// TwinCAT 3 PLC project SAmpleVisionRefactoringSimple
// ProgramVersion: 3.1.4024.0
// libraries:
//   Tc2_Standard, * (Beckhoff Automation GmbH)
//   Tc2_System, * (Beckhoff Automation GmbH)
//   Tc3_Module, * (Beckhoff Automation GmbH)
// project tree:
//   DUTs/ LED1904.TcDUT
//   DUTs/Vision/ ST_CenterPosition.TcDUT, ST_ColorSimularity.TcDUT, ST_Conture.TcDUT, ST_PositionBounds.TcDUT, ST_PositionDeviation.TcDUT, ST_PositionXY.TcDUT, ST_ThresholdData.TcDUT
//   GVLs/ Globale_Definitionen.TcGVL, Globale_Kamera_Variablen.TcGVL
//   / PlcTask.TcTTO
//   POUs/ Camera.TcPOU, MAIN.TcPOU
// (motion and I/O tree: see PLC project plc1)
// real-time tasks:
//   TASK PlcTask: cycle T#10ms, priority 20, ADS port 350
//   TASK PlcTask1: cycle T#10ms, priority 21, ADS port 351
//   TASK PlcTask2: cycle T#10ms, priority 22, ADS port 352

CONFIGURATION SAmpleVisionRefactoringSimple
    RESOURCE PLC ON TwinCAT3
        TASK PlcTask(INTERVAL := T#10ms, PRIORITY := 22);
        PROGRAM MAIN WITH PlcTask : MAIN;
    END_RESOURCE
END_CONFIGURATION

// ---- DUTs/LED1904.TcDUT
TYPE LED1904 :
STRUCT
	bInput1:BOOL;
	bInput2:BOOL;
	bInput3:BOOL;
	bInput4:BOOL;
	bDiag1:BOOL;
	bDiag2:BOOL;
	bDiag3:BOOL;
	bDiag4:BOOL;
END_STRUCT
END_TYPE

// ---- DUTs/Vision/ST_CenterPosition.TcDUT
TYPE ST_CenterPosition :
STRUCT
  Input : ST_PositionXY;
  Diagnose : ST_PositionXY;
END_STRUCT
END_TYPE

// ---- DUTs/Vision/ST_ColorSimularity.TcDUT
TYPE ST_ColorSimularity :
STRUCT
	aRefColor :	TcVnPoint3_LREAL;
	aRefColorGreen : TcVnPoint3_LREAL	:= [130, 230, 0];
	aRefColorRed : TcVnPoint3_LREAL	:= [255, 255, 255];
	aRefColorPrismError :	TcVnPoint3_LREAL := [135, 150, 105];
	fVariance :	REAL := 0.10;
	fLuminanceWeight :	REAL := 0.1;
END_STRUCT
END_TYPE

// ---- DUTs/Vision/ST_Conture.TcDUT
TYPE ST_Conture :
STRUCT
	fAreaMin : REAL;		(*Mindestfläche der zufindenden LED*)
	fAreaMax : REAL;		(*Mindestfläche der zufindenden LED*)
	fHeightMin : REAL;		(*Mindesthöhe der zufindenden LED*)
	fHeightMax : REAL;		(*Maximalhöhe der zufindenden LED*)
	fWidthMax : REAL;		(*Maximalhöhe der zufindenden LED*)
END_STRUCT
END_TYPE

// ---- DUTs/Vision/ST_PositionBounds.TcDUT
TYPE ST_PositionBounds :
STRUCT
  stDeviation : ST_PositionDeviation; 
	aCenterReferenceCoordinatesXY	: ARRAY  [1..8] OF TcVnPoint2_REAL;
  aCenterPosition : ARRAY[1..4] OF ST_CenterPosition;  
END_STRUCT
END_TYPE

// ---- DUTs/Vision/ST_PositionDeviation.TcDUT
TYPE ST_PositionDeviation :
STRUCT
  nLower : UINT;
	nUpper : UINT;
END_STRUCT
END_TYPE

// ---- DUTs/Vision/ST_PositionXY.TcDUT
TYPE ST_PositionXY :
STRUCT
  X : REAL;
  Y : REAL;
END_STRUCT
END_TYPE

// ---- DUTs/Vision/ST_ThresholdData.TcDUT
TYPE ST_ThresholdData :
STRUCT
	fThreshold : LREAL;	(* fixed threshold (unused if dynamic thresholding is selected) *)
	fMaxValue :	LREAL;	(* maximum pixel value *)
END_STRUCT
END_TYPE

// ---- GVLs/Globale_Definitionen.TcGVL
{attribute 'Tc2GvlVarNames'}
VAR_GLOBAL
	FileName: STRING := 'C:\TwinSAFE\TestErgebnisse\EL1904\TestLog_EL1904_';
	StartUp_Wait_Time: TIME := t#3s;
	ShutDown_Wait_Time : TIME := T#1S;
	Kamera_Wait_Time: TIME := T#2S;
	Prisma_Wait_Time:  TIME := T#3S;
	Seriell_Wait_Time: TIME := T#1S;
	KameraBeleuchtungFaktorWarteZeit:UINT:=8;
	Kopfzeile: STRING(255);
	TesterArray: ARRAY[0..7] OF STRING ;
	EtherCATAmsNetID: T_AmsNetId := '172.16.3.218.2.1';
	EL1904port: T_AmsPort := 1024;
	EL6900port: T_AmsPort := 1010;
	OutputWait_Time: TIME := t#5s;
	Color_Rot : DWORD := 16#000000FF;
	Color_Gruen : DWORD := 16#00007F00;
	Color_Weiss : DWORD := 16#00FFFFFF;
	Color_Visu : DWORD := 16#00FFFFFF;
	VoltagePowerContacts20Vunder : UINT := 21300; (* 0V = 0, 30V = 32767  1092 pro Volt  20V = 21845*)
	VoltagePowerContacts20Vover : UINT := 22300; (* 0V = 0, 30V = 32767  1092 pro Volt  20V = 21845*)
	VoltagePowerContacts24Vunder : UINT := 25900; (* 0V = 0, 30V = 32767  1092 pro Volt  24V = 26213*)
	VoltagePowerContacts24Vover : UINT := 26700; (* 0V = 0, 30V = 32767  1092 pro Volt  24V = 26213*)
	VoltagePowerContacts30Vunder : UINT := 32200; (* 0V = 0, 30V = 32767  1092 pro Volt  30V = 32767*)
	VoltagePowerContacts30Vover : UINT := 32767; (* 0V = 0, 30V = 32767  1092 pro Volt  30V = 32767*)
	LogFileSerialNumber: UDINT;
	Artikel : UDINT := 70931;
//	SafetyProg1: T_MaxString := 'C:\TwinSAFE\Programm\EL\Automated_EL1904\1_SafetyProgramCRC';
//	SafetyCRC1: WORD := 17617;
	SafetyProg65534: T_MaxString := 'C:\TwinSAFE\Programm\EL\Automated_EL1904\65534_SafetyProgramCRC';
	SafetyCRC65534: WORD := 65346;
END_VAR

// ---- GVLs/Globale_Kamera_Variablen.TcGVL
{attribute 'qualified_only'}
VAR_GLOBAL
	//TestVariablen
	bStopStepPrismaDetection:BOOL:=FALSE;
	bStopStepAllLedOn:BOOL:=FALSE;
	bEinrichtBetrieb:BOOL:=FALSE;
	bNextStepEinrichtbetrieb:BOOL:=FALSE;
	bPrismaOk:BOOL:=FALSE;
	bPrismaNotOK:BOOL:=FALSE;
	
	//Kamera aktiv
	bKameraAktiv:BOOL:=TRUE;
	
	//erkannte LEDs
	bLED_TermXOn		: ARRAY  [1..8] OF LED1904;
	iDetectedLED			: INT:=0;
	iStartDetectedLED		: INT:=1;
	
	// Color Simularity
//	aRefColor					:	TcVnPoint3_LREAL;
//	aRefColorGreen				:	TcVnPoint3_LREAL	:= [130, 230, 0];
//	aRefColorRed				:	TcVnPoint3_LREAL	:= [255, 255, 255];
//	aRefColorPrismError			:	TcVnPoint3_LREAL	:= [135, 150, 105];
//	fVariance					:	REAL := 0.10;
//	fLuminanceWeight			:	REAL := 0.1;
  stColorSimularity : ST_ColorSimularity;
  
  
	
	//Threshold
  stThreshold : ST_ThresholdData; 
  stThresholdGreenLed : ST_ThresholdData := (fThreshold := 10, fMaxValue := 255); 
  stThresholdRedLed : ST_ThresholdData := (fThreshold := 15, fMaxValue := 255); 
  stThresholdPrism : ST_ThresholdData := (fThreshold := 185, fMaxValue := 255); 
	
	//Konturen zeichnen
  stConture : ST_Conture := (fAreaMin := 1200,fAreaMax := 3000, fHeightMin := 30, fHeightMax := 70, fWidthMax:= 70 );
  stContureLED : ST_Conture := (fAreaMin := 1200,fAreaMax := 3000, fHeightMin := 30, fHeightMax := 70, fWidthMax:= 90 );
  stConturePrisma : ST_Conture := (fAreaMin := 450,fAreaMax := 900, fHeightMin := 20, fHeightMax := 70, fWidthMax:= 70 );
	
	// Positionsgrenzen
//	uiLowerPosDeviation:UINT:=10;
//	uiUpperPosDeviation:UINT:=10;
//	aCenterReferenceCoordinatesXY	: ARRAY  [1..8] OF TcVnPoint2_REAL;
//	CenterXPosInput1:REAL:=46;
//	CenterYPosInput1:REAL:=36;
//	CenterXPosInput2:REAL:=119;
//	CenterYPosInput2:REAL:=33;
//	CenterXPosInput3:REAL:=46;
//	CenterYPosInput3:REAL:=87;
//	CenterXPosInput4:REAL:=120;
//	CenterYPosInput4:REAL:=87;
//	CenterXPosDiag1:REAL:=46;
//	CenterYPosDiag1:REAL:=139;
//	CenterXPosDiag2:REAL:=114;
//	CenterYPosDiag2:REAL:=137;
//	CenterXPosDiag3:REAL:=45;
//	CenterYPosDiag3:REAL:=192;
//	CenterXPosDiag4:REAL:=124;
//	CenterYPosDiag4:REAL:=192;
  
  stPositionBounds : ST_PositionBounds;


//PositionBounds.aCenterPosition[1].Diagnose.X
  
  
	// Region of Interrest
	nXposPrisma			:	UDINT:=1514;
	nYposPrisma			:	UDINT:=892;
	nROIWidth			:	UDINT:=170;
	nROIHeight			:	UDINT:=220;
	
	// Beleuchtung EL2595
	bLedOn AT%Q* :BOOL;
	uiOutputCurrent AT%Q*:UINT;
	bLedReset AT%Q*:BOOL;
	bLedWarning AT%I*:BOOL;
	bLedError AT%I*:BOOL;	
	uiOutputCurrentEinrichtbertieb:UINT:=300;
END_VAR

// ---- POUs/MAIN.TcPOU
PROGRAM MAIN
VAR
END_VAR

END_PROGRAM

// ---- POUs/Camera.TcPOU
PROGRAM Camera
VAR
	
  hr : HRESULT;
  fbCameraControl :	FB_VN_GevCameraControl; //SymbolInitialization  verlinken!
	eState : ETcVnCameraState;
	
	ipImgIn :	ITcVnImage;
	ipImgRoi :   ITcVnImage;
	ipImgRotated :   ITcVnImage;
	ipImgConvertColorSpace : 	ITcVnImage;
	ipImgColorSimilarity :	ITcVnImage;
	ipImgThreshold :	ITcVnImage;
	ipImgResult :	ITcVnImage;
	
	ipImg_Eingangsbild : ITcVnDisplayableImage;
	ipImg_Ausgeschnitten : ITcVnDisplayableImage;
	ipImg_Gedreht :	ITcVnDisplayableImage;
	ipImg_Farbbild : ITcVnDisplayableImage;
	ipImg_Farbauswahl :	ITcVnDisplayableImage;
	ipImg_Schwellwert_Farbauswahl :	ITcVnDisplayableImage;
	ipImg_Ergebnis :	ITcVnDisplayableImage;
	
	
	// Region of Interrest
	nXposTerm1 : UDINT;
	nYposTerm1 : UDINT;
	nROIWidth :	UDINT;
	nROIHeight : UDINT;
	
	// Get Center 
	aCenterCoordinatesXY : ARRAY[1..8] OF TcVnPoint2_REAL;
	
	aWhite : TcVnVector4_LREAL :=	[255,255,255];
	aBlack : TcVnVector4_LREAL :=	[0,0,0];
	aRed : TcVnVector4_LREAL := 	[255,0,0];
	aGreen : TcVnVector4_LREAL :=	[0,255,0];
	aBlue :	TcVnVector4_LREAL :=	[0,0,255];
	aOrange :	TcVnVector4_LREAL :=	[255,150,0];
END_VAR

VAR
  // Init
  bInitPositionBoundsDone : BOOL := FALSE;
  nClearByteLength : UDINT;
END_VAR

// Init
InitPositionBounds(bInitPositionBoundsDone, Globale_Kamera_Variablen.stPositionBounds);


// Position zum Zuschneiden des Prismas aus der Visu übergeben
nXposTerm1 := Globale_Kamera_Variablen.nXposPrisma;
nYposTerm1 := Globale_Kamera_Variablen.nYposPrisma;
nROIWidth := Globale_Kamera_Variablen.nROIWidth;
nROIHeight := Globale_Kamera_Variablen.nROIHeight;

// Kamera Kontroll Status Maschine
eState := fbCameraControl.GetState();
//eState := fbFileSource.GetState();

CASE eState OF
	
  TCVN_CS_INITIAL, TCVN_CS_OPENING, TCVN_CS_OPENED, TCVN_CS_STARTACQUISITION:
    hr := fbCameraControl.StartAcquisition();
	
  TCVN_CS_ACQUIRING:
    hr := fbCameraControl.GetCurrentImage(ipImgIn);
	
    IF SUCCEEDED(hr) AND ipImgIn <> 0 THEN
      VisionLedDetecting(); 		(*Methoden Aufruf*)
    
      hr := F_VN_TransformIntoDisplayableImage(ipImgIn, ipImg_Eingangsbild, S_OK);
      hr := F_VN_TransformIntoDisplayableImage(ipImgRoi, ipImg_Ausgeschnitten, S_OK);
      hr := F_VN_TransformIntoDisplayableImage(ipImgRotated, ipImg_Gedreht, S_OK);
      hr := F_VN_TransformIntoDisplayableImage(ipImgConvertColorSpace, ipImg_Farbbild, S_OK);
      hr := F_VN_TransformIntoDisplayableImage(ipImgColorSimilarity, ipImg_Farbauswahl, S_OK);
      hr := F_VN_TransformIntoDisplayableImage(ipImgThreshold, ipImg_Schwellwert_Farbauswahl, S_OK);
      hr := F_VN_TransformIntoDisplayableImage(ipImgResult, ipImg_Ergebnis, S_OK);
      
    END_IF

  // Freigeben der Bilder sonst kann es zum Page Fault kommen
    Tc3_Module.FW_SafeRelease(ADR(ipImgIn));
    Tc3_Module.FW_SafeRelease(ADR(ipImgRoi));
    Tc3_Module.FW_SafeRelease(ADR(ipImgRotated));
    Tc3_Module.FW_SafeRelease(ADR(ipImgConvertColorSpace));
    Tc3_Module.FW_SafeRelease(ADR(ipImgColorSimilarity));
    Tc3_Module.FW_SafeRelease(ADR(ipImgThreshold));
    Tc3_Module.FW_SafeRelease(ADR(ipImgResult));

  TCVN_CS_ERROR:
    //hr := fbFileSource.Reset();
    hr := fbCameraControl.Reset();
    
  END_CASE

//Positionen der Mittelpunktskoordinaten aus der Visu übernehmen
GetCenterPositionFromVisu(Globale_Kamera_Variablen.stPositionBounds);
	
//Detectiere LEDs	
//Diag1 LED
Globale_Kamera_Variablen.iStartDetectedLED:=1;
DetectLedCoordinate(
    nStartDetectedLED:= Globale_Kamera_Variablen.iStartDetectedLED, 
    nDetectedLED:= Globale_Kamera_Variablen.iDetectedLED, 
    nLedNumber:= 5, 
    aCenterCoordinatesXY:= aCenterCoordinatesXY[Globale_Kamera_Variablen.iStartDetectedLED], 
    stPositionBounds:= Globale_Kamera_Variablen.stPositionBounds, 
    Detected:= Globale_Kamera_Variablen.bLED_TermXOn[1].bDiag1);

//Diag2 LED
Globale_Kamera_Variablen.iStartDetectedLED:=1;
DetectLedCoordinate(
    nStartDetectedLED:= Globale_Kamera_Variablen.iStartDetectedLED, 
    nDetectedLED:= Globale_Kamera_Variablen.iDetectedLED, 
    nLedNumber:= 6, 
    aCenterCoordinatesXY:= aCenterCoordinatesXY[Globale_Kamera_Variablen.iStartDetectedLED], 
    stPositionBounds:= Globale_Kamera_Variablen.stPositionBounds, 
    Detected:= Globale_Kamera_Variablen.bLED_TermXOn[1].bDiag2);

//Diag3 LED
Globale_Kamera_Variablen.iStartDetectedLED:=1;
DetectLedCoordinate(
    nStartDetectedLED:= Globale_Kamera_Variablen.iStartDetectedLED, 
    nDetectedLED:= Globale_Kamera_Variablen.iDetectedLED, 
    nLedNumber:= 7, 
    aCenterCoordinatesXY:= aCenterCoordinatesXY[Globale_Kamera_Variablen.iStartDetectedLED], 
    stPositionBounds:= Globale_Kamera_Variablen.stPositionBounds, 
    Detected:= Globale_Kamera_Variablen.bLED_TermXOn[1].bDiag3);


//Diag4 LED
Globale_Kamera_Variablen.iStartDetectedLED:=1;
DetectLedCoordinate(
    nStartDetectedLED:= Globale_Kamera_Variablen.iStartDetectedLED, 
    nDetectedLED:= Globale_Kamera_Variablen.iDetectedLED, 
    nLedNumber:= 8, 
    aCenterCoordinatesXY:= aCenterCoordinatesXY[Globale_Kamera_Variablen.iStartDetectedLED], 
    stPositionBounds:= Globale_Kamera_Variablen.stPositionBounds, 
    Detected:= Globale_Kamera_Variablen.bLED_TermXOn[1].bDiag4);

//Input1 LED
Globale_Kamera_Variablen.iStartDetectedLED:=1;
DetectLedCoordinate(
    nStartDetectedLED:= Globale_Kamera_Variablen.iStartDetectedLED, 
    nDetectedLED:= Globale_Kamera_Variablen.iDetectedLED, 
    nLedNumber:= 1, 
    aCenterCoordinatesXY:= aCenterCoordinatesXY[Globale_Kamera_Variablen.iStartDetectedLED], 
    stPositionBounds:= Globale_Kamera_Variablen.stPositionBounds, 
    Detected:= Globale_Kamera_Variablen.bLED_TermXOn[1].bInput1);

//Input2 LED
Globale_Kamera_Variablen.iStartDetectedLED:=1;
DetectLedCoordinate(
    nStartDetectedLED:= Globale_Kamera_Variablen.iStartDetectedLED, 
    nDetectedLED:= Globale_Kamera_Variablen.iDetectedLED, 
    nLedNumber:= 2, 
    aCenterCoordinatesXY:= aCenterCoordinatesXY[Globale_Kamera_Variablen.iStartDetectedLED], 
    stPositionBounds:= Globale_Kamera_Variablen.stPositionBounds, 
    Detected:= Globale_Kamera_Variablen.bLED_TermXOn[1].bInput2);

//Input3 LED
Globale_Kamera_Variablen.iStartDetectedLED:=1;
DetectLedCoordinate(
    nStartDetectedLED:= Globale_Kamera_Variablen.iStartDetectedLED, 
    nDetectedLED:= Globale_Kamera_Variablen.iDetectedLED, 
    nLedNumber:= 3, 
    aCenterCoordinatesXY:= aCenterCoordinatesXY[Globale_Kamera_Variablen.iStartDetectedLED], 
    stPositionBounds:= Globale_Kamera_Variablen.stPositionBounds, 
    Detected:= Globale_Kamera_Variablen.bLED_TermXOn[1].bInput3);

//Input4 LED
Globale_Kamera_Variablen.iStartDetectedLED:=1;
DetectLedCoordinate(
    nStartDetectedLED:= Globale_Kamera_Variablen.iStartDetectedLED, 
    nDetectedLED:= Globale_Kamera_Variablen.iDetectedLED, 
    nLedNumber:= 4, 
    aCenterCoordinatesXY:= aCenterCoordinatesXY[Globale_Kamera_Variablen.iStartDetectedLED], 
    stPositionBounds:= Globale_Kamera_Variablen.stPositionBounds, 
    Detected:= Globale_Kamera_Variablen.bLED_TermXOn[1].bInput4);

// CenterCoordinatesXY Rücksetzen, damit neuer durchlauf starten kann.
IF ( Globale_Kamera_Variablen.iStartDetectedLED >= 0) AND (Globale_Kamera_Variablen.iStartDetectedLED < 7)  THEN
  nClearByteLength := TO_UDINT(TO_INT( SIZEOF(aCenterCoordinatesXY[1])) * (8 - Globale_Kamera_Variablen.iStartDetectedLED));
  memset(ADR(aCenterCoordinatesXY[Globale_Kamera_Variablen.iStartDetectedLED + 1]), 0, nClearByteLength);
  END_IF

METHOD PRIVATE ClearCenterCorodinatesXY : HRESULT
VAR_INPUT
  iStartDetectedLED : INT;
END_VAR

IF iStartDetectedLED < 0 OR iStartDetectedLED > 8 THEN
  ClearCenterCorodinatesXY := Tc3_Module.E_FAIL; //ADSERR_DEVICE_INVALIDPARM
  RETURN;
END_IF
END_METHOD

METHOD PRIVATE DetectLedCoordinate : HRESULT
VAR_INPUT
  nStartDetectedLED : INT;
  nDetectedLED : INT;
  nLedNumber : INT;
  aCenterCoordinatesXY : TcVnPoint2_REAL;
  stPositionBounds : ST_PositionBounds; 
  Detected : REFERENCE TO BOOL;
END_VAR

Detected := FALSE;	

FOR nStartDetectedLED:=1 TO nDetectedLED BY 1 DO
  IF aCenterCoordinatesXY[0] > stPositionBounds.aCenterReferenceCoordinatesXY[nLedNumber][0] - stPositionBounds.stDeviation.nLower
    AND aCenterCoordinatesXY[0] < stPositionBounds.aCenterReferenceCoordinatesXY[nLedNumber][0] + stPositionBounds.stDeviation.nUpper
    AND aCenterCoordinatesXY[1] > stPositionBounds.aCenterReferenceCoordinatesXY[nLedNumber][1] - stPositionBounds.stDeviation.nLower
    AND aCenterCoordinatesXY[1] < stPositionBounds.aCenterReferenceCoordinatesXY[nLedNumber][1] + stPositionBounds.stDeviation.nUpper THEN
      Detected := TRUE;	
    END_IF
  END_FOR  
DetectLedCoordinate := Tc3_Module.S_OK;
END_METHOD

METHOD PRIVATE GetCenterPositionFromVisu : HRESULT
VAR_INPUT
  stPositionBounds : REFERENCE TO ST_PositionBounds;
END_VAR

stPositionBounds.aCenterReferenceCoordinatesXY[1][0]:= stPositionBounds.aCenterPosition[1].Input.X;
stPositionBounds.aCenterReferenceCoordinatesXY[1][1]:= stPositionBounds.aCenterPosition[1].Input.y;
stPositionBounds.aCenterReferenceCoordinatesXY[2][0]:= stPositionBounds.aCenterPosition[2].Input.X;
stPositionBounds.aCenterReferenceCoordinatesXY[2][1]:= stPositionBounds.aCenterPosition[2].Input.y;
stPositionBounds.aCenterReferenceCoordinatesXY[3][0]:= stPositionBounds.aCenterPosition[3].Input.X;
stPositionBounds.aCenterReferenceCoordinatesXY[3][1]:= stPositionBounds.aCenterPosition[3].Input.y;
stPositionBounds.aCenterReferenceCoordinatesXY[4][0]:= stPositionBounds.aCenterPosition[4].Input.X;
stPositionBounds.aCenterReferenceCoordinatesXY[4][1]:= stPositionBounds.aCenterPosition[4].Input.y;
stPositionBounds.aCenterReferenceCoordinatesXY[5][0]:= stPositionBounds.aCenterPosition[1].Diagnose.X;
stPositionBounds.aCenterReferenceCoordinatesXY[5][1]:= stPositionBounds.aCenterPosition[1].Diagnose.Y;
stPositionBounds.aCenterReferenceCoordinatesXY[6][0]:= stPositionBounds.aCenterPosition[2].Diagnose.X;
stPositionBounds.aCenterReferenceCoordinatesXY[6][1]:= stPositionBounds.aCenterPosition[2].Diagnose.Y;
stPositionBounds.aCenterReferenceCoordinatesXY[7][0]:= stPositionBounds.aCenterPosition[3].Diagnose.X;
stPositionBounds.aCenterReferenceCoordinatesXY[7][1]:= stPositionBounds.aCenterPosition[3].Diagnose.Y;
stPositionBounds.aCenterReferenceCoordinatesXY[8][0]:= stPositionBounds.aCenterPosition[4].Diagnose.X;
stPositionBounds.aCenterReferenceCoordinatesXY[8][1]:= stPositionBounds.aCenterPosition[4].Diagnose.Y;

GetCenterPositionFromVisu := Tc3_Module.S_OK;
END_METHOD

METHOD PRIVATE InitPositionBounds : HRESULT
VAR_INPUT
  bInitPositionBoundsDone : BOOL;
  PositionBounds : REFERENCE TO ST_PositionBounds;
END_VAR

IF bInitPositionBoundsDone THEN RETURN; END_IF

PositionBounds.stDeviation.nLower :=10;
PositionBounds.stDeviation.nUpper :=10;
PositionBounds.aCenterPosition[1].Input.X := 46;
PositionBounds.aCenterPosition[1].Input.Y := 36;
PositionBounds.aCenterPosition[2].Input.X := 119;
PositionBounds.aCenterPosition[2].Input.Y := 33;
PositionBounds.aCenterPosition[3].Input.X := 46;
PositionBounds.aCenterPosition[3].Input.Y := 87;
PositionBounds.aCenterPosition[4].Input.X := 120;
PositionBounds.aCenterPosition[4].Input.Y := 87;

PositionBounds.aCenterPosition[1].Diagnose.X := 46;
PositionBounds.aCenterPosition[1].Diagnose.Y := 139;
PositionBounds.aCenterPosition[2].Diagnose.X := 114;
PositionBounds.aCenterPosition[2].Diagnose.Y := 137;
PositionBounds.aCenterPosition[3].Diagnose.X := 45;
PositionBounds.aCenterPosition[3].Diagnose.Y := 192;
PositionBounds.aCenterPosition[4].Diagnose.X := 124;
PositionBounds.aCenterPosition[4].Diagnose.Y := 192;

bInitPositionBoundsDone := TRUE;

InitPositionBounds  := Tc3_Module.S_OK;
END_METHOD

METHOD PRIVATE VisionLedDetecting 
VAR
	ipImgWork :	ITcVnImage;
	
	ipContours :	ITcVnContainer;
	ipContour :	ITcVnContainer;
	ipForwardIterator :	ITcVnForwardIterator;
	aContourOffset : TcVnPoint;
	
	fArea :	LREAL;
	stRect : TcVnRotatedRectangle;
	
	
END_VAR

//	Region of Interrest
hr := F_VN_CopyImage(ipImgIn, ipImgRoi, hr);
hr:= F_VN_SetRoi( nXposTerm1, nYposTerm1, nROIWidth, nROIHeight,ipImgRoi ,hr);

// Rotate Image
hr:=F_VN_RotateImage(ipImgRoi,ipImgRotated,TCVN_RA_180_DEG,hr);
hr := F_VN_CopyImage(ipImgRotated, ipImgRotated, hr);

// Color Space
hr := F_VN_ConvertColorSpace(ipImgRotated (*ipImgRoi*)(*ipImgIn*), ipImgWork, ETcVNColorSpaceTransform.TCVN_CST_BAYER_GR_TO_BGR , hr); //TCVN_CST_BAYER_GR_TO_RGB TCVN_CST_BAYER_BG_TO_RGB Liegt daran wie das Bild abgeschnitten wurde
hr := F_VN_CopyImage(ipImgWork, ipImgConvertColorSpace, hr);

//Color Simularity
hr := F_VN_ReferenceColorSimilarityExp_TcVnVector3_LREAL(ipImgWork, ipImgWork, Globale_Kamera_variablen.stColorSimularity.aRefColor, Globale_Kamera_Variablen.stColorSimularity.fVariance, Globale_Kamera_Variablen.stColorSimularity.fLuminanceWeight, hr);
hr := F_VN_CopyImage(ipImgWork, ipImgColorSimilarity, hr);

//Threshold
hr := Tc3_Vision.F_VN_Threshold(ipImgWork, ipImgWork, Globale_Kamera_Variablen.stThreshold.fThreshold, Globale_Kamera_Variablen.stThreshold.fMaxValue, ETcVnThresholdType.TCVN_TT_BINARY, hr);
hr := F_VN_CopyImage(ipImgWork, ipImgThreshold, hr);


// Contours
hr := F_VN_FindContoursExp(ipImgWork, ipContours, ETcVnContourRetrievalMode.TCVN_CRM_CONNECTED_COMPONENTS, ETcVnContourApproximationMethod.TCVN_CAM_SIMPLE, aContourOffset,hr);


IF SUCCEEDED(hr) AND ipContours <> 0 THEN
	hr := F_VN_GetForwardIterator(ipContours, ipForwardIterator, hr);
	
	// Create an Image to display the results
	hr := F_VN_ConvertColorSpace(ipImgRotated(*ipImgRoi*) (*ipImgIn*), ipImgWork, ETcVNColorSpaceTransform.TCVN_CST_BAYER_GR_TO_BGR, hr);
	
	Globale_Kamera_Variablen.iDetectedLED := 0;
	
	WHILE SUCCEEDED(hr) AND ipForwardIterator.CheckIfEnd() = S_FALSE DO
		
		hr := F_VN_GetContainer(ipForwardIterator, ipContour, hr);
		hr := F_VN_IncrementIterator(ipForwardIterator, hr);
		

		// Finding Criteria to Filter the Contours
		//============================================
		
		// (2) Area and Rectangle Shape		
		hr := Tc3_Vision.F_VN_ContourArea(ipContour, fArea, hr);
		IF fArea > Globale_Kamera_Variablen.stConture.fAreaMin THEN 
			
			//hr := F_VN_DetermineEnclosingRectangle(ipContour, stRect, hr);
			hr := Tc3_Vision.F_VN_EnclosingRectangle(ipContour, stRect, hr);
			
			Globale_Kamera_Variablen.iDetectedLED:= Globale_Kamera_Variablen.iDetectedLED + 1;// Falls Bild noch nicht zugeschnitten eventuell auskommentieren wegen Exception
	 
			aCenterCoordinatesXY[Globale_Kamera_Variablen.iDetectedLED]:=stRect.aCenter; // Falls Bild noch nicht zugeschnitten eventuell auskommentieren wegen Exception
			
			// Prüfen ob "Quadratisch" 									
			IF stRect.stSize.fHeight > Globale_Kamera_Variablen.stConture.fHeightMin AND stRect.stSize.fHeight < Globale_Kamera_Variablen.stConture.fHeightMax AND stRect.stSize.fWidth < Globale_Kamera_Variablen.stConture.fWidthMax THEN 
				hr := F_VN_DrawContours(ipContour, -1, ipImgWork, aGreen, 2, hr);				
			ELSIF fArea > Globale_Kamera_Variablen.stConture.fAreaMax THEN
				hr := F_VN_DrawContours(ipContour, -1, ipImgWork, aOrange, 2, hr);
			ELSE
				hr := F_VN_DrawContours(ipContour, -1, ipImgWork, aRed, 2, hr);
			END_IF
			
		END_IF
					
		//F_VN_ReleaseInterface(ipContour);
		Tc3_Module.FW_SafeRelease(ADR(ipContour));
	END_WHILE

END_IF

hr := F_VN_CopyImage(ipImgWork, ipImgResult, hr);


// Release all Interface Pointer
Tc3_Module.FW_SafeRelease(ADR(ipContours));
Tc3_Module.FW_SafeRelease(ADR(ipForwardIterator));
Tc3_Module.FW_SafeRelease(ADR(ipImgWork));
END_METHOD

END_PROGRAM
